TYPE ST_TECStatus :
STRUCT
	//Parameters
	diTemp1	:	DINT;
	diSetPoint	:	DINT;
	diPercentOut	:	DINT;
	diCurrent	:	DINT;
	xOutputOn	:	BOOL;
	
	//Alarms
	xHiTemp	:	BOOL;
	xLoTemp	:	BOOL;
	xCompCtrlAlrm	:	BOOL;
	xOverCurrent	:	BOOL;
	xOpenInput1		:	BOOL;
	xOpenInput2		:	BOOL;
	xDriverLowVoltage	:	BOOL;
	
	
	//Interface Diagnosis
xStatusValid	:	BOOL;
sReply	:	STRING;

END_STRUCT
END_TYPE

(* stored: Version 1.1.0.1, ProductVersion 3.1.0.24
   DUT ST_TECStatus: Id {df12744f-874c-412c-aed2-7be14a84a0c5} *)
